FUNCTION_BLOCK I_VP1 (* Vehicle Position 1 *)
  (* Standard: ISO 11783-7; Classification: PGN 65267; Function: Vehicle Position 1; Description: Copyright (c) 2024 HR Agrartechnik GmbH This program and the accompanying materials are made available under the terms of the Eclipse Public License 2.0 which is available at https://www.eclipse.org/legal/epl-2.0/ SPDX-License-Identifier: EPL-2.0 https://docs.ms-muc-docs.de/projects/isobus-other-docs/de/latest/PGN/PGN_65267.html *)
  (* Version 1.0, 07.02.2025, Moritz Ortmeier, HR Agrartechnik GmbH *)
  PACKAGE isobus::tecu;
  IMPORT eclipse4diac::core::TypeHash;
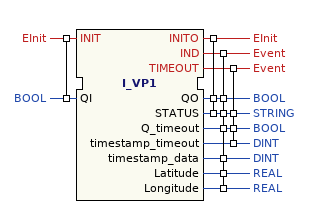
  EVENT_INPUT
    INIT : EInit WITH QI; (* Service Initialization *)
  END_EVENT
  EVENT_OUTPUT
    INITO : EInit WITH QO, STATUS; (* Initialization Confirm *)
    IND WITH QO, timestamp_data, Latitude, Longitude, STATUS, Q_timeout; (* Indication from Resource *)
    TIMEOUT WITH timestamp_timeout, STATUS, Q_timeout;
  END_EVENT
  VAR_INPUT
    QI : BOOL; (* Event Input Qualifier *)
  END_VAR
  VAR_OUTPUT
    QO : BOOL; (* Event Output Qualifier *)
    STATUS : STRING;
    Q_timeout : BOOL;
    timestamp_timeout : DINT;
    timestamp_data : DINT;
    Latitude : REAL; {SET_ATTRIBUTE(SPN, 584)} {SET_ATTRIBUTE(SP_Name, 'Latitude')} {SET_ATTRIBUTE(SP_Position_In_PG, '1-4')} {SET_ATTRIBUTE(SP_Length, 4)} (* 4 Bytes *) {SET_ATTRIBUTE(Scaling, )} {SET_ATTRIBUTE(Offset, -210)} (* deg offset *) {SET_ATTRIBUTE(Link, 'https://docs.ms-muc-docs.de/projects/isobus-other-docs/de/latest/PGN/PGN_65267.html#spn-584-latitude')}
    Longitude : REAL; {SET_ATTRIBUTE(SPN, 585)} {SET_ATTRIBUTE(SP_Name, 'Longitude')} {SET_ATTRIBUTE(SP_Position_In_PG, '5-8')} {SET_ATTRIBUTE(SP_Length, 4)} (* 4 bytes *) {SET_ATTRIBUTE(Scaling, '')} {SET_ATTRIBUTE(Offset, -210)} (* deg offset *) {SET_ATTRIBUTE(Link, 'https://docs.ms-muc-docs.de/projects/isobus-other-docs/de/latest/PGN/PGN_65267.html#spn-585-longitude')}
  END_VAR
END_FUNCTION_BLOCK
